# EPICS substitutions: db/Beckhoff_3XXX/ecmcEL3174_0to20mA.substitutions
#Actually the scalinging is between 0..21.474mA (see manual)
file "ecmc_analogInput-chX.template"
{
  pattern {CH_ID, ESLO, EOFF, EGU, PREC, LOW, LOLO, HIGH, HIHI, HYST, LLSV, LSV, HSV, HHSV}
          {01, "${_ESLO=6.5535447249E-4}", "${_EOFF=0}", "${_EGU=mA}", "${_PREC=3}", 0, -1, 20, 21, 0, "MAJOR", "MINOR", "MINOR", "MAJOR"}
          {02, "${_ESLO=6.5535447249E-4}", "${_EOFF=0}", "${_EGU=mA}", "${_PREC=3}", 0, -1, 20, 21, 0, "MAJOR", "MINOR", "MINOR", "MAJOR"}
          {03, "${_ESLO=6.5535447249E-4}", "${_EOFF=0}", "${_EGU=mA}", "${_PREC=3}", 0, -1, 20, 21, 0, "MAJOR", "MINOR", "MINOR", "MAJOR"}
          {04, "${_ESLO=6.5535447249E-4}", "${_EOFF=0}", "${_EGU=mA}", "${_PREC=3}", 0, -1, 20, 21, 0, "MAJOR", "MINOR", "MINOR", "MAJOR"}
}

file "ecmc_status_analog-chX.template"
{
  pattern {CH_ID, KEY }
          {01,    "AI"}
          {02,    "AI"}
          {03,    "AI"}
          {04,    "AI"}
}
